FUNCTION_BLOCK INTERNAL FB_FileHelper_Tests EXTENDS FB_TestSuite

Test01_ValidateReferences();

METHOD Test01_ValidateReferences
VAR_INPUT
END_VAR
TcUnit.TEST('Test01_ValidateReferences');

AssertTrue(FileHelper.Directory <> 0, 'Directory property is not valid!');
AssertTrue(FileHelper.File <> 0, 'File property is not valid!');
AssertTrue(FileHelper.Path <> 0, 'Path property is not valid!');

TcUnit.TEST_FINISHED();
END_METHOD

END_FUNCTION_BLOCK

(* stored: Version 1.1.0.1, ProductVersion 3.1.4024.14
   POU FB_FileHelper_Tests: Id {9989709f-a59d-0c20-3f70-73122c507dbf}, SpecialFunc None
   Method Test01_ValidateReferences: Id {0d42137c-8623-0088-35c6-235fb63fc1b1} *)
